# EPICS autosave request: pmac/pmacController_settings.req
$(P):COORDINATE_SYS_GROUP
